{attribute addProperty BoxType "KL3362"}
{attribute addProperty Id "Channel_1Channel_C961C78600Channel_2Channel_C961C78600"}
{attribute addProperty CRC "1467776686"}
{attribute addProperty SizeInBites "0"}
{attribute addProperty SizeInBytes "0"}
TYPE KL3362_577C7EAE :
STRUCT
	{attribute addProperty Name "Channel_1"}
	Channel_1 : Channel_C961C786;
	{attribute addProperty Name "Channel_2"}
	Channel_2 : Channel_C961C786;
END_STRUCT
END_TYPE

(* stored: Version 1.2.0.0, ProductVersion 3.1.4024.9
   DUT KL3362_577C7EAE: Id {59098112-d9c8-423b-9ad8-5cd467559ad6} *)
